FUNCTION_BLOCK MONGO_DB_CT
  {SET_ATTRIBUTE(OpcUa, SERVICE)}
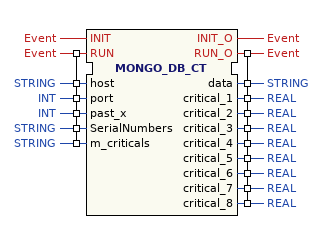
  EVENT_INPUT
    INIT;
    RUN WITH host, port, past_x, SerialNumbers, m_criticals; {SET_ATTRIBUTE(OpcUa, Method)}
  END_EVENT
  EVENT_OUTPUT
    INIT_O;
    RUN_O WITH data, critical_1, critical_2, critical_3, critical_4, critical_5, critical_6, critical_7, critical_8;
  END_EVENT
  VAR_INPUT
    host : STRING; {SET_ATTRIBUTE(OpcUa, Variable.RUN)}
    port : INT; {SET_ATTRIBUTE(OpcUa, Variable.RUN)}
    past_x : INT; {SET_ATTRIBUTE(OpcUa, Variable.RUN)}
    SerialNumbers : STRING; {SET_ATTRIBUTE(OpcUa, Variable.RUN)}
    m_criticals : STRING; {SET_ATTRIBUTE(OpcUa, Variable.RUN)}
  END_VAR
  VAR_OUTPUT
    data : STRING; {SET_ATTRIBUTE(OpcUa, Variable.RUN)}
    critical_1 : REAL; {SET_ATTRIBUTE(OpcUa, Variable.RUN)}
    critical_2 : REAL; {SET_ATTRIBUTE(OpcUa, Variable.RUN)}
    critical_3 : REAL; {SET_ATTRIBUTE(OpcUa, Variable.RUN)}
    critical_4 : REAL; {SET_ATTRIBUTE(OpcUa, Variable.RUN)}
    critical_5 : REAL; {SET_ATTRIBUTE(OpcUa, Variable.RUN)}
    critical_6 : REAL; {SET_ATTRIBUTE(OpcUa, Variable.RUN)}
    critical_7 : REAL; {SET_ATTRIBUTE(OpcUa, Variable.RUN)}
    critical_8 : REAL; {SET_ATTRIBUTE(OpcUa, Variable.RUN)}
  END_VAR
END_FUNCTION_BLOCK
